FUNCTION_BLOCK ABSTRACT POU_3
VAR_INPUT
END_VAR
VAR_OUTPUT
END_VAR
VAR
END_VAR

END_FUNCTION_BLOCK

(* stored: Version 1.1.0.1, ProductVersion 3.1.4024.12
   POU POU_3: Id {ab6a28e3-5fe5-47df-8b86-a2465f1734ed}, SpecialFunc None *)
